// TIA Portal V20 export
TYPE "zp_CITIData"
// stored: Namespace CITI_Logic
   STRUCT
      EoC { S7_SetPoint := 'True'} : "CITI_Logic.zp_CITIEoC";
      CoS : "CITI_Logic.zp_CITICoS";
      TradeCall { S7_SetPoint := 'True'} : "CITI_Logic.zp_CITITradeCalls";
      FaultString { S7_SetPoint := 'True'} : String[200];   // Fault String to PMC
      Machine_Loading : Bool;   // Machine Loading Bit
      Machine_Unloading : Bool;   // Machine Unloading Bit
      Machine_Processing : Bool;   // Machine Processing Bit
      Shift_Reset : Bool;   // Shift Reset
      Clock_Sync : Bool;   // Clock Sync from PMC
      Dry_Cycle_Mode : Bool;   // Dry Cycle
      CITI_DryCycle_Blocker : Bool;   // CITI Dry Cycle Blocker
      Control_Power_On : Bool;   // Control Power On
      IT_Heartbeat : Bool;   // IT Heartbeat
      Write_Day : SInt;   // Sync Day
      Write_Month : SInt;   // Sync Month
      Write_Year : SInt;   // Sync Year
      ShiftNumber : SInt;   // Shift Number from PMC
      Current_Cycle_Time : DInt;   // Current Cycle Time
   END_STRUCT;
END_TYPE
